// TIA Portal V21 export
DATA_BLOCK "DB621"   // DB621
TITLE = DB619
{ S7_Optimized_Access := 'TRUE' }
// CIP BUTTONS DB
// stored: AutoNumber false, MemoryReserve 0
   VAR
      Start : Bool;
   END_VAR
   VAR RETAIN
      MainPopup1Ack : Bool;
      MainPopup2Ack : Bool;
   END_VAR
BEGIN
END_DATA_BLOCK
